(* Schneider Machine Expert - Basic project Timer 1, file version 1.7.0.0 *)
(* ProjectInformations: Name=New project *)

HARDWARE
  Cpu 0: TM221M16R/G
  EthernetConfiguration: NetworkName=M221, IpAllocationMode=FixedAddress, IpAddress=0.0.0.0, SubnetMask=0.0.0.0
  SerialLineConfiguration: Baud=Baud19200, Parity=ParityEven, DataBits=DataBits8, StopBits=StopBits1, PhysicalMedium=PhysicalMediumRs485, TransmissionMode=TransmissionModeModbusRtu, SlaveId=1, Addressing=SlaveAddressing
  MastTask: UsePeriodScanMode=false, PeriodScan=100
  FastTask: Period=255
  CpuBehavior: StartingMode=StartAsPreviousState, AutoSaveRamOnEeprom=true, WatchdogPeriod=250

SYMBOLS  (address, symbol, comment, settings)
  %TM0        "T1 2""  [Preset=20, Base=OneHundredMilliSeconds]
  %TM1        "T2 2""  [Preset=20, Base=OneHundredMilliSeconds]
  %I0.0       "S1"
  %Q0.0       "L1"
  %Q0.1       "L2"

POU New POU
  (* SectionNumber=1 *)

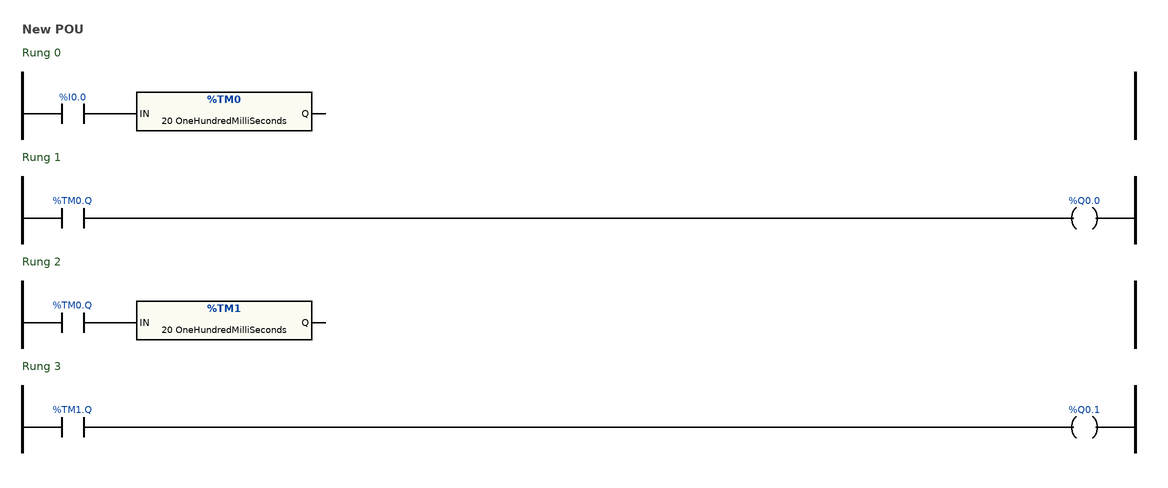

// Rung 0
  BLK %TM0
  LD %I0.0
  IN
  END_BLK
  // as ST:
  //   %TM0(IN := %I0.0);

// Rung 1
  LD %TM0.Q
  ST %Q0.0
  // as ST:
  //   %Q0.0 := %TM0.Q;

// Rung 2
  BLK %TM1
  LD %TM0.Q
  IN
  END_BLK
  // as ST:
  //   %TM1(IN := %TM0.Q);

// Rung 3
  LD %TM1.Q
  ST %Q0.1
  // as ST:
  //   %Q0.1 := %TM1.Q;
